Fanuc KAREL source: ko00079.KL

-- PROVISIONAL review KL for V940-1; original PC SHA256 8c72f3949d97af809c65b4001f1b39d17376c1230200fd356da620a567e1799d
-- Incomplete behavior may be omitted. Consult companion uncertainty JSON. Do not deploy.
PROGRAM KO00079
%NOLOCKGROUP
BEGIN
  -- V9_ZERO_TABLE_METADATA_HINT layout=0002_ascii; no indexed target words; source/name/runtime held
  -- UNRESOLVED_PC offsets 5-12; opcodes 9D,23
  -- UNRESOLVED_PC offsets 17-66; opcodes 27,22,1C,27,49,7E,AD,22,31,7E,4A
  -- UNRESOLVED_PC offsets 71-75; opcodes 7F
END KO00079
